FUNCTION_BLOCK FACTORY_IO_SORTING
  {SET_ATTRIBUTE(OpcUa, DEVICE.SENSOR)}
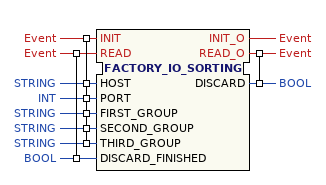
  EVENT_INPUT
    INIT WITH HOST, PORT, FIRST_GROUP, SECOND_GROUP, THIRD_GROUP;
    READ WITH DISCARD_FINISHED;
  END_EVENT
  EVENT_OUTPUT
    INIT_O;
    READ_O WITH DISCARD;
  END_EVENT
  VAR_INPUT
    HOST : STRING; {SET_ATTRIBUTE(OpcUa, Constant.RUN)}
    PORT : INT; {SET_ATTRIBUTE(OpcUa, Constant.RUN)}
    FIRST_GROUP : STRING; {SET_ATTRIBUTE(OpcUa, Constant.RUN)}
    SECOND_GROUP : STRING; {SET_ATTRIBUTE(OpcUa, Constant.RUN)}
    THIRD_GROUP : STRING; {SET_ATTRIBUTE(OpcUa, Constant.RUN)}
    DISCARD_FINISHED : BOOL; {SET_ATTRIBUTE(OpcUa, Variable.RUN)}
  END_VAR
  VAR_OUTPUT
    DISCARD : BOOL; {SET_ATTRIBUTE(OpcUa, Variable.RUN)}
  END_VAR
END_FUNCTION_BLOCK
